FUNCTION F_AddChannelToHeader : BOOL
// Adds data about our channel to the header
VAR_IN_OUT
    stHeader: DUT_Header_NW;
    stChannel: DUT_Channel_NW;
END_VAR

IF stChannel.channel = 0 THEN
    F_AddChannelToHeader := FALSE;
ELSE
    stHeader.channelMask := stHeader.channelMask + SHL(1, stChannel.channel - 1);
    IF stChannel.error > 0 THEN
        stHeader.errorMask := stHeader.errorMask + SHL(1, stChannel.channel - 1);
    END_IF
    F_AddChannelToHeader := TRUE;
END_IF

END_FUNCTION

(* stored: Version 1.1.0.1, ProductVersion 3.1.4022.18
   POU F_AddChannelToHeader: Id {959519f1-ba9d-4157-89b1-d9ff7bcd8738}, SpecialFunc None *)
